// TwinCAT 3 PLC project PlcSample_IpcDiag
// ProgramVersion: 3.1.4020.4
// libraries:
//   Tc2_Standard, * (Beckhoff Automation GmbH)
//   Tc2_System, * (Beckhoff Automation GmbH)
//   Tc3_IPCDiag, * (Beckhoff Automation GmbH)
//   Tc3_Module, * (Beckhoff Automation GmbH)
// project tree:
//   DUTs/ E_State.TcDUT, stIPCDiag.TcDUT, ST_MDP_Error.TcDUT, ST_ServiceTransfer_DeleteFile.TcDUT
//   GVLs/ GVL.TcGVL
//   / PlcTask.TcTTO (not stored)
//   POUs/ FB_Change_IP.TcPOU, FB_Change_AmsNetId.TcPOU, FB_IPC_DeleteFile.TcPOU, FB_ReadBiosInfo.TcPOU, MAIN.TcPOU
// real-time tasks:
//   TASK PlcTask: cycle T#10ms, priority 20, ADS port 350

// ---- DUTs/E_State.TcDUT
{attribute 'qualified_only'}
TYPE E_State :
(
	Init := 0,
	ReadOnce,
	ReadPeriodically,
	Error,
	
	Idle,
	DeleteFolder,
	ReadOnce_CpuUsage,
	ReadOnce_CpuTemperature,
	ReadOnce_SrnMainboard,
	ReadOnce_SrnIPC,
	ReadBios,
	Write_DHCP,
	Write_IPAddr,
	SetAmsNetId
);
END_TYPE

// ---- DUTs/stIPCDiag.TcDUT
TYPE stIPCDiag :
	
STRUCT
	//Read Once---------------------------------------------------------------------------
	sIPCDeviceName		: STRING(39);
	sIPCSerialNumber: STRING;
	
	nCpuFreq		: UDINT;
	nCpuUsage		: UINT;
	
	nTcBuild		: UINT;
	sTC_Version		: STRING;
	
	aNIC_Name		: ARRAY[1..IpcDiagnostics.cMaxNumberList] OF STRING(79);	// array in order to receive info of up to three network ports (NICs)
	aNIC_IPv4Address: ARRAY[1..IpcDiagnostics.cMaxNumberList] OF STRING(39);	// array in order to receive info of up to three network ports (NICs)
	aNIC_DHCP		: ARRAY[1..IpcDiagnostics.cMaxNumberList] OF BOOL;		// array in order to receive info of up to three network ports (NICs)
	nNIC_ModuleCnt	: UINT;
	
	nMassStg_NoDrives			:UINT;	
	aMassStg_DriveList_DriveName:ARRAY[1..IpcDiagnostics.cMaxNumberList] OF STRING(79);
 
	sMdpVersion		: STRING;
	nBootCnt		: UDINT;
	
	//Periodische Daten--------------------------------------------------------------------
	nCpuTemperature	: INT;							// [°C]; should be read periodically	
	
END_STRUCT

END_TYPE

// ---- DUTs/ST_MDP_Error.TcDUT
{attribute 'pack_mode' := '1'}
TYPE ST_MDP_Error :
STRUCT
	mdp_state : BYTE;
	padding	  : BYTE;
	mdp_error : DWORD;
END_STRUCT
END_TYPE

// ---- DUTs/ST_ServiceTransfer_DeleteFile.TcDUT
{attribute 'pack_mode' := '1'}
TYPE ST_ServiceTransfer_DeleteFile :
STRUCT
	cbFileName : DWORD;
	bRecursive : DWORD; // Error in documentation
	s_filename : STRING;
END_STRUCT
END_TYPE

// ---- GVLs/GVL.TcGVL
{attribute 'qualified_only'}
VAR_GLOBAL
	amsNetId : T_AmsNetId  := '';
END_VAR

// ---- POUs/FB_Change_IP.TcPOU
FUNCTION_BLOCK FB_Change_IP
VAR_IN_OUT
	modules : ST_IPCDiag_ModuleList;
END_VAR
VAR_INPUT
	ipAddr : STRING;
	bExec 	 : BOOL;
END_VAR
VAR_OUTPUT
	bBusy		: BOOL;
	bError		: BOOL;
	mdp_error	: ST_MDP_Error;
	nErrId		: HRESULT;
	//errMsg		: Tc3_IPCDiag.I_TcMessage;
END_VAR
VAR
	state 			: INT := 0;
	eErrorState 	: INT;
	i 				: UINT;
	modId 			: INT := -1;
	mdpIdx			: WORD;
	mdp_status		: BYTE;
	bExecFlank		: BOOL;
	fbWriteParam	: FB_IPCDiag_WriteParameterByMdpIdx;
	fbReadParam		: FB_IPCDiag_ReadParameterByMdpIdx;

END_VAR

IF NOT bExec AND bExecFlank THEN
		bExecFlank := FALSE;
END_IF



CASE state OF

0: // Idle
	bBusy := FALSE;
	// steigende flanke
	IF bExec AND NOT bExecFlank THEN
		bExecFlank := TRUE;
		state := 1;
		bBusy := TRUE;
	END_IF
1: // find module
	
	// Find Module Idx of File System Object
	WHILE i <= modules.nModules OR modId = - 1 DO
		IF modules.aModules[i].eModType = E_IPCDiag_ModuleType.NIC THEN // File System Object
			modId := modules.aModules[i].nModId;
		END_IF
		i := i + 1;
	END_WHILE
	state := 2;
	
2: // Execute delete folder
	mdpIdx := 16#8001 + DINT_TO_WORD(SHL(modId, 4));
	
	
	fbWriteParam(
		bExecute:= TRUE, 
		nIndex:= mdpIdx,
		nFlags:= 0, //  
		nSubIndex:= 2, // Trigger / Write // BAUSTELLE
		pBuffer:= ADR(ipAddr), 
		nBufferSize:= INT_TO_UINT(LEN(ipAddr)),
	);
		
	IF NOT fbWriteParam.bBusy THEN
		IF fbWriteParam.bError THEN
			bError 	:= TRUE;
			nErrId	:= fbWriteParam.hrErrorCode;
			//errMsg	: fbWriteParam.ipErrorMessage;
			eErrorState := state;
			state := 99;
		ELSE
			bError 	:= FALSE;
			state := 0;
		END_IF
		fbWriteParam(bExecute:=FALSE);
	END_IF
	
	
9: // Error state
	;
END_CASE

END_FUNCTION_BLOCK

// ---- POUs/FB_Change_AmsNetId.TcPOU
FUNCTION_BLOCK FB_Change_AmsNetId
VAR_IN_OUT
	modules : ST_IPCDiag_ModuleList;
END_VAR
VAR_INPUT
	amsNetId : STRING;
	bExec 	 : BOOL;
END_VAR
VAR_OUTPUT
	bBusy		: BOOL;
	bError		: BOOL;
	mdp_error	: ST_MDP_Error;
	nErrId		: HRESULT;
	//errMsg		: Tc3_IPCDiag.I_TcMessage;
END_VAR
VAR
	state 			: INT := 0;
	eErrorState 	: INT;
	i 				: UINT;
	modId 			: INT := -1;
	mdpIdx			: WORD;
	mdp_status		: BYTE;
	bExecFlank		: BOOL;
	fbWriteParam	: FB_IPCDiag_WriteParameterByMdpIdx;
	//fbReadParam		: FB_IPCDiag_ReadParameterByMdpIdx;

END_VAR

IF NOT bExec AND bExecFlank THEN
		bExecFlank := FALSE;
END_IF



CASE state OF

0: // Idle
	bBusy := FALSE;
	// steigende flanke
	IF bExec AND NOT bExecFlank THEN
		bExecFlank := TRUE;
		state := 1;
		bBusy := TRUE;
	END_IF
1: // find module
	
	// Find Module Idx of File System Object
	WHILE i <= modules.nModules OR modId = - 1 DO
		IF modules.aModules[i].eModType = E_IPCDiag_ModuleType.TwinCAT THEN // File System Object
			modId := modules.aModules[i].nModId;
		END_IF
		i := i + 1;
	END_WHILE
	state := 2;
	
2: // Execute delete folder
	mdpIdx := 16#8001 + DINT_TO_WORD(SHL(modId, 4));
	
	fbWriteParam(
		bExecute:= TRUE, 
		nIndex:= mdpIdx,
		nFlags:= 0, //  
		nSubIndex:= 4, // Ams Net Id
		pBuffer:= ADR(amsNetId), 
		nBufferSize:= INT_TO_UINT(LEN(amsNetId)),
	);
		
	IF NOT fbWriteParam.bBusy THEN
		IF fbWriteParam.bError THEN
			bError 	:= TRUE;
			nErrId	:= fbWriteParam.hrErrorCode;
			//errMsg	: fbWriteParam.ipErrorMessage;
			eErrorState := state;
			state := 99;
		ELSE
			bError 	:= FALSE;
			state := 0;
		END_IF
		fbWriteParam(bExecute:=FALSE);
	END_IF
	
	
9: // Error state
	;
END_CASE

END_FUNCTION_BLOCK

// ---- POUs/FB_IPC_DeleteFile.TcPOU
FUNCTION_BLOCK FB_IPC_DeleteFile
VAR_IN_OUT
	modules : ST_IPCDiag_ModuleList;
END_VAR
VAR_INPUT
	filename : STRING;
	bExec 	 : BOOL;
END_VAR
VAR_OUTPUT
	bBusy		: BOOL;
	bError		: BOOL;
	mdp_error	: ST_MDP_Error;
	nErrId		: HRESULT;
	//errMsg		: Tc3_IPCDiag.I_TcMessage;
END_VAR
VAR
	state 			: INT := 0;
	eErrorState 	: INT;
	i 				: UINT;
	modId 			: INT := -1;
	mdpIdx			: WORD;
	mdp_status		: BYTE;
	bExecFlank		: BOOL;
	st_del_file		: ST_ServiceTransfer_DeleteFile;
	fbWriteParam	: FB_IPCDiag_WriteParameterByMdpIdx;
	fbReadParam		: FB_IPCDiag_ReadParameterByMdpIdx;
END_VAR

IF NOT bExec AND bExecFlank THEN
		bExecFlank := FALSE;
END_IF



CASE state OF

0: // Idle
	bBusy := FALSE;
	// steigende flanke
	IF bExec AND NOT bExecFlank THEN
		bExecFlank := TRUE;
		state := 1;
		bBusy := TRUE;
	END_IF
1: // find module
	
	// Find Module Idx of File System Object
	WHILE i <= modules.nModules OR modId = - 1 DO
		IF modules.aModules[i].eModType = E_IPCDiag_ModuleType.FileSystemObject THEN // File System Object
			modId := modules.aModules[i].nModId;
		END_IF
		i := i + 1;
	END_WHILE
	state := 2;
	
2: // Execute delete folder
	mdpIdx := 16#B004 + DINT_TO_WORD(SHL(modId, 4));
	
	st_del_file.cbFileName := INT_TO_DWORD(LEN(fileName)) ;
	st_del_file.bRecursive := BOOL_TO_DWORD(FALSE);
	st_del_file.s_filename := filename;
	
	fbWriteParam(
		bExecute:= TRUE, 
		nIndex:= mdpIdx,
		nFlags:= 0, //  
		nSubIndex:= 1, // Trigger / Write 
		pBuffer:= ADR(st_del_file), 
		nBufferSize:= INT_TO_DWORD(LEN(fileName)) + SIZEOF(st_del_file.bRecursive) + SIZEOF(st_del_file.cbFileName),
		sNetId := modules.sNetId
	);
		
	IF NOT fbWriteParam.bBusy THEN
		IF fbWriteParam.bError THEN
			bError 	:= TRUE;
			nErrId	:= fbWriteParam.hrErrorCode;
			//errMsg	: fbWriteParam.ipErrorMessage;
			eErrorState := state;
			state := 99;
		ELSE
			bError 	:= FALSE;
			state := 3;
		END_IF
		fbWriteParam(bExecute:=FALSE);
	END_IF
	
3: // Get state of operation

	fbReadParam(
		bExecute:= TRUE, 
		nIndex:= mdpIdx, 
		nFlags:= 0, 
		nSubIndex:= 2, 
		pBuffer:= ADR(mdp_status), 
		nBufferSize:= SIZEOF(mdp_status),
		sNetId := modules.sNetId
	);
	IF NOT fbReadParam.bBusy THEN
		IF fbReadParam.bError THEN
			bError 	:= TRUE;
			nErrId	:= fbWriteParam.hrErrorCode;
			//errMsg	: fbWriteParam.ipErrorMessage;
			eErrorState := state;
			state := E_State.Error;
		ELSE
			
			IF mdp_status = 3 THEN
				bError 	:= TRUE;
				state := 4;
			ELSE
				bError 	:= FALSE;
				bBusy := FALSE;
				state := 0;
			END_IF
		END_IF
		fbReadParam(bExecute:=FALSE);
	END_IF

4: // Get error code of operation

	fbReadParam(
		bExecute:= TRUE, 
		nIndex:= mdpIdx, 
		nFlags:= 0, 
		nSubIndex:= 3, 
		pBuffer:= ADR(mdp_error), 
		nBufferSize:= SIZEOF(mdp_error), 
		sNetId := modules.sNetId
	);
	IF NOT fbReadParam.bBusy THEN
			bError 	:= TRUE;
		IF fbReadParam.bError THEN
			nErrId	:= fbWriteParam.hrErrorCode;
			//errMsg	: fbWriteParam.ipErrorMessage;
			eErrorState := state;
			state := 99;
		ELSE
			state := 0;
		END_IF
		fbReadParam(bExecute:=FALSE);
	END_IF
	
9: // Error state
	;
END_CASE

END_FUNCTION_BLOCK

// ---- POUs/FB_ReadBiosInfo.TcPOU
FUNCTION_BLOCK FB_ReadBiosInfo
VAR_IN_OUT
	modules : ST_IPCDiag_ModuleList;
END_VAR
VAR_INPUT
	bExec 	 : BOOL;
END_VAR
VAR_OUTPUT
	bBusy		: BOOL;
	bError		: BOOL;
	mdp_error	: ST_MDP_Error;
	nErrId		: HRESULT;
END_VAR
VAR
	state 			: INT := 0;
	eErrorState 	: INT;
	i 				: UINT;
	modId 			: INT := -1;
	mdpIdx			: WORD;
	mdp_status		: BYTE;
	bExecFlank		: BOOL;
	fbWriteParam	: FB_IPCDiag_WriteParameterByMdpIdx;
	fbReadParam		: FB_IPCDiag_ReadParameterByMdpIdx;
	
	bios_major		: USINT;
	bios_minor 		: USINT; 
	n_bytesRead		: UDINT;
END_VAR

IF NOT bExec AND bExecFlank THEN
		bExecFlank := FALSE;
END_IF



CASE state OF

0: // Idle
	bBusy := FALSE;
	// steigende flanke
	IF bExec AND NOT bExecFlank THEN
		bExecFlank := TRUE;
		state := 1;
		bBusy := TRUE;
	END_IF
1: // find module
	
	// Find Module Idx of File System Object
	WHILE i <= modules.nModules OR modId = - 1 DO
		IF modules.aModules[i].eModType = E_IPCDiag_ModuleType.Mainboard THEN // File System Object
			modId := modules.aModules[i].nModId;
		END_IF
		i := i + 1;
	END_WHILE
	state := 2;
	
2: // Bios Major
	mdpIdx := 16#8002 + DINT_TO_WORD(SHL(modId, 4));
	

	fbReadParam(
		bExecute:= TRUE, 
		nIndex:= mdpIdx, 
		nFlags:= 0, 
		nSubIndex:= 2, // Bios Major
		pBuffer:= ADR(bios_major), 
		nBufferSize:= SIZEOF(bios_major),  
		nCount=> n_bytesRead);
	IF NOT fbReadParam.bBusy THEN
		IF fbReadParam.bError THEN
			bError 	:= TRUE;
			nErrId	:= fbReadParam.hrErrorCode;
			//errMsg	: fbWriteParam.ipErrorMessage;
			eErrorState := state;
			state := 99;
		ELSE
			bError 	:= FALSE;
			state := 3;
		END_IF
		fbReadParam(bExecute:=FALSE);
	END_IF

3: // Bios Minor

	fbReadParam(
		bExecute:= TRUE, 
		nIndex:= mdpIdx, 
		nFlags:= 0, 
		nSubIndex:= 3, // Bios Minor
		pBuffer:= ADR(bios_minor), 
		nBufferSize:= SIZEOF(bios_minor),  
		nCount=> n_bytesRead);
	IF NOT fbReadParam.bBusy THEN
		IF fbReadParam.bError THEN
			bError 	:= TRUE;
			nErrId	:= fbReadParam.hrErrorCode;
			//errMsg	: fbWriteParam.ipErrorMessage;
			eErrorState := state;
			state := 99;
		ELSE
			bError 	:= FALSE;
			state := 0;
		END_IF
		fbReadParam(bExecute:=FALSE);
	END_IF
9: // Error state
	;
END_CASE

END_FUNCTION_BLOCK

// ---- POUs/MAIN.TcPOU
PROGRAM MAIN
VAR
	
	//sNetId			: T_AmsNetID := '5.69.55.236.1.1';
	fb_file_delete	: FB_IPC_DeleteFile;
	fb_change_ip	: FB_Change_IP;
	fb_setAmsNetUd  : FB_Change_AmsNetId;
	fb_readBios		: FB_ReadBiosInfo;
	fbDiagRegister  : FB_IPCDiag_Register; // := (sNetId:=sNetId);
	moduleList		: ST_IPCDiag_ModuleList;
	eState			: E_State := E_State.Init;
	eErrorState 	: E_State;
	hrGetValue		: HRESULT;	
	
	modId			: INT := -1; // 0 is a valid value
	mdpIdx			: WORD;
	i				: UINT;
	test : ST_IPCDiag_Module;
	fileName		: STRING := 'C:\test';
	
	
	
END_VAR

CASE eState OF
	
E_State.Init: 
	
	IF NOT fbDiagRegister.bBusy THEN
		fbDiagRegister(bExecute:=TRUE,); // need to be executed once
	ELSE
		fbDiagRegister(bExecute:=FALSE);
	END_IF
	
	IF NOT fbDiagRegister.bBusy THEN
		IF fbDiagRegister.bError THEN
			eErrorState := eState;
			eState := E_State.Error;
		ELSE
			//eState := E_State.DeleteFolderExec;
			//eState := E_State.Write_IPAddr;
			//eState := E_State.SetAmsNetId;
			eState := E_State.ReadBios;
			moduleList := fbDiagRegister.stModuleList;
		END_IF
	END_IF
	

E_State.Idle:
	;	
	
	
	
E_State.DeleteFolder:
	fb_file_delete(
		modules:= moduleList, 
		filename:= fileName, 
		bExec:= TRUE
		);
	IF NOT fb_file_delete.bBusy THEN
		IF fb_file_delete.bError THEN
			eErrorState := eState;
			eState := E_State.Error;
		ELSE
			eErrorState := E_State.Idle;
		END_IF
		fb_file_delete(modules:= moduleList, bExec:=FALSE);
	END_IF
	
E_State.Write_IPAddr:
	
	fb_change_ip(
		modules:= moduleList, 
		ipAddr:= '192.168.1.1', 
		bExec:= TRUE
		);
	IF NOT fb_change_ip.bBusy THEN
		IF fb_change_ip.bError THEN
			eErrorState := eState;
			eState := E_State.Error;
		ELSE
			eErrorState := E_State.Idle;
		END_IF
		fb_change_ip(modules:= moduleList, bExec:=FALSE);
	END_IF
	
E_State.SetAmsNetId:
	fb_setAmsNetUd(
		modules:=moduleList, 
		amsNetId:= '5.80.201.232.1.1', 
		bExec:= TRUE, 
	 );
	 IF NOT fb_setAmsNetUd.bBusy THEN
		IF fb_setAmsNetUd.bError THEN
			eErrorState := eState;
			eState := E_State.Error;
		ELSE
			eState := E_State.Idle;
		END_IF
		fb_setAmsNetUd(modules:= moduleList, bExec:=FALSE);
	END_IF
	;

E_State.ReadBios:
	fb_readBios(
		modules:=moduleList, 
		bExec:= TRUE 
	);
	IF NOT fb_readBios.bBusy THEN
		IF fb_readBios.bError THEN
			eErrorState := eState;
			eState := E_State.Error;
		ELSE
			eState := E_State.Idle;
		END_IF
		fb_readBios(modules:= moduleList, bExec:=FALSE);
	END_IF
E_State.Error:
	;
END_CASE

END_PROGRAM
